// TIA Portal project "Project0" (V16)

(* hardware
DEVICE "S7-1200 station_1"  S7-1200 Station
   slot 0: "Rack_0"  S7-1200 Rack  Rack  V1.0
   slot 1: "PLC_1"  CPU 1214C AC/DC/Rly  6ES7 214-1BG40-0XB0  V4.2
*)

// ===== PLC "PLC_1"  CPU 1214C AC/DC/Rly =====

VAR_GLOBAL   // PLC tag table "Default tag table"
   ""START"" AT %I0.0 : Bool;
   ""STOP"" AT %I0.1 : Bool;
   ""MODE"" AT %I0.2 : Bool;
   ""SENSOR_1"" AT %I0.3 : Bool;
   ""SENSOR_2"" AT %I0.4 : Bool;
   ""SENSOR_3"" AT %I0.5 : Bool;
   ""SENSOR_4"" AT %I0.6 : Bool;
   ""SENSOR_5"" AT %I0.7 : Bool;
   ""SENSOR_6"" AT %I1.0 : Bool;
   ""SENSOR_7"" AT %I1.1 : Bool;
   ""SENSOR_8"" AT %I1.2 : Bool;
   ""Sim"" AT %I1.3 : Bool;
   ""CONVEYOR_BELT_1"" AT %Q0.0 : Bool;
   ""CONVEYOR_BELT_2"" AT %Q0.1 : Bool;
   ""CONVEYOR_BELT_3"" AT %Q0.2 : Bool;
   ""CONVEYOR_BELT_4_L"" AT %Q0.3 : Bool;
   ""CONVEYOR_BELT_4_R"" AT %Q0.4 : Bool;
   ""CONTAINER_1_FULL"" AT %Q0.5 : Bool;
   ""CONTAINER_2_FULL"" AT %Q0.6 : Bool;
END_VAR